// TIA Portal V16 export
// export: Created 2021-05-25T16:14:40.8525101Z, ExportSetting WithDefaults, DisplayName Totally Integrated Automation Portal, DisplayVersion V16, DisplayName TIA Portal Version Control Interface, DisplayVersion V16, DisplayName TIA Portal Openness, DisplayVersion V16, DisplayName STEP 7 Professional, DisplayVersion V16, DisplayName STEP 7 Safety, DisplayVersion V16, DisplayName WinCC Unified SCADA Engineering System, DisplayVersion V16
DATA_BLOCK "dbSystemAlarms"   // DB105
{ S7_Optimized_Access := 'FALSE'; DB_Accessible_From_OPC_UA := 'FALSE' }
VERSION : 0.1
// stored: AutoNumber false, DBAccessibleFromOPCUA false, IsOnlyStoredInLoadMemory false, IsWriteProtectedInAS false
   VAR
      SysAlm : Array[1..1024] of Bool;
      EthAlm : Array[1..128] of Bool;
      DPAlm : Array[1..16, 1..16] of DWord;
   END_VAR
BEGIN
   SysAlm[1..128] := FALSE;
   EthAlm[1..128] := FALSE;
   DPAlm[1,1..16] := 16#0000_0000;
   DPAlm[2,1..16] := 16#0000_0000;
   DPAlm[3,1..16] := 16#0000_0000;
   DPAlm[4,1..16] := 16#0000_0000;
   DPAlm[5,1..16] := 16#0000_0000;
   DPAlm[6,1..16] := 16#0000_0000;
   DPAlm[7,1..16] := 16#0000_0000;
   DPAlm[8,1..16] := 16#0000_0000;
   DPAlm[9,1..16] := 16#0000_0000;
   DPAlm[10,1..16] := 16#0000_0000;
   DPAlm[11,1..16] := 16#0000_0000;
   DPAlm[12,1..16] := 16#0000_0000;
   DPAlm[13,1..16] := 16#0000_0000;
   DPAlm[14,1..16] := 16#0000_0000;
   DPAlm[15,1..16] := 16#0000_0000;
   DPAlm[16,1..16] := 16#0000_0000;
END_DATA_BLOCK
